(* CoDeSys 2.3.9.28 project: Aula08_ex2.pro *)
(* Libraries: Standard.lib 27.1.09 11:27:38, Util.lib 27.1.09 11:27:38, IecSfc.lib 24.11.08 08:07:15, SysLibTime.lib 27.1.09 11:27:38, SysTaskInfo.lib 24.11.08 08:07:15, SYSLIBCALLBACK.LIB 27.1.09 11:27:38 *)

(* PLC configuration (modules and I/O channels)
Hexswitch AT %IB0 [HexSwitch] rotary switch 0 = STOP, 1-15 = RUN
IOModules [CPX_MASTER] node 0, in %IB4 out %QB0
  8DI/8DO [CPX-8DI_8DO_Multi_I_O_module_1] node 0, in %IB4 out %QB0 {StringParam = 4,8,1,8,1; ByteParam = 7; ByteParam = 81; ByteParam = 0; ByteParam = 0; ByteParam = 0; ByteParam = 0; ByteParam = 0; IdleStateParam = 0; IdleModeParam = 255; IdleStateParam = 0; IdleModeParam = 255; IdleStateParam = 0; IdleModeParam = 255; IdleStateParam = 0; IdleModeParam = 255}
    AT %IB4 [ByteInput] -
    AT %QB0 [ByteOutput] -
  8DI/8DO [CPX-8DI_8DO_Multi_I_O_module_1] node 1, in %IB8 out %QB4 {StringParam = 4,8,1,8,1; ByteParam = 7; ByteParam = 81; ByteParam = 0; ByteParam = 0; ByteParam = 0; ByteParam = 0; ByteParam = 0; IdleStateParam = 0; IdleModeParam = 255; IdleStateParam = 0; IdleModeParam = 255; IdleStateParam = 0; IdleModeParam = 255; IdleStateParam = 0; IdleModeParam = 255}
    AT %IB8 [ByteInput] -
    AT %QB4 [ByteOutput] -
*)

(* Global variable list: Global_Variables *)
VAR_GLOBAL

	START AT %IX2.0 : BOOL;
	STOP AT %IX2.1 : BOOL;
	S1 AT %IX2.2 : BOOL;
	S2 AT %IX2.3 : BOOL;
	S3 AT %IX2.4 : BOOL;
	S4 AT %IX2.5 : BOOL;

	M1 AT %QX0.0 : BOOL;
	LP AT %QX0.1 : BOOL;
	C1 AT %QX0.2 : BOOL;
	C2 AT %QX0.3 : BOOL;

	MEM : BOOL;
	MEM2 : BOOL;
	MEM3: BOOL;
	MEM4: BOOL;
	MEM5: BOOL;

	T : TON;

END_VAR

(* POU PLC_PRG, LD *)
PROGRAM PLC_PRG
VAR

	T1: TON;
END_VAR
VAR (* helpers for the ST form of the networks *)
	_p1 : BOOL;
	_p2 : BOOL;
	_p3 : BOOL;
	_p4 : BOOL;
	_p5 : BOOL;
END_VAR
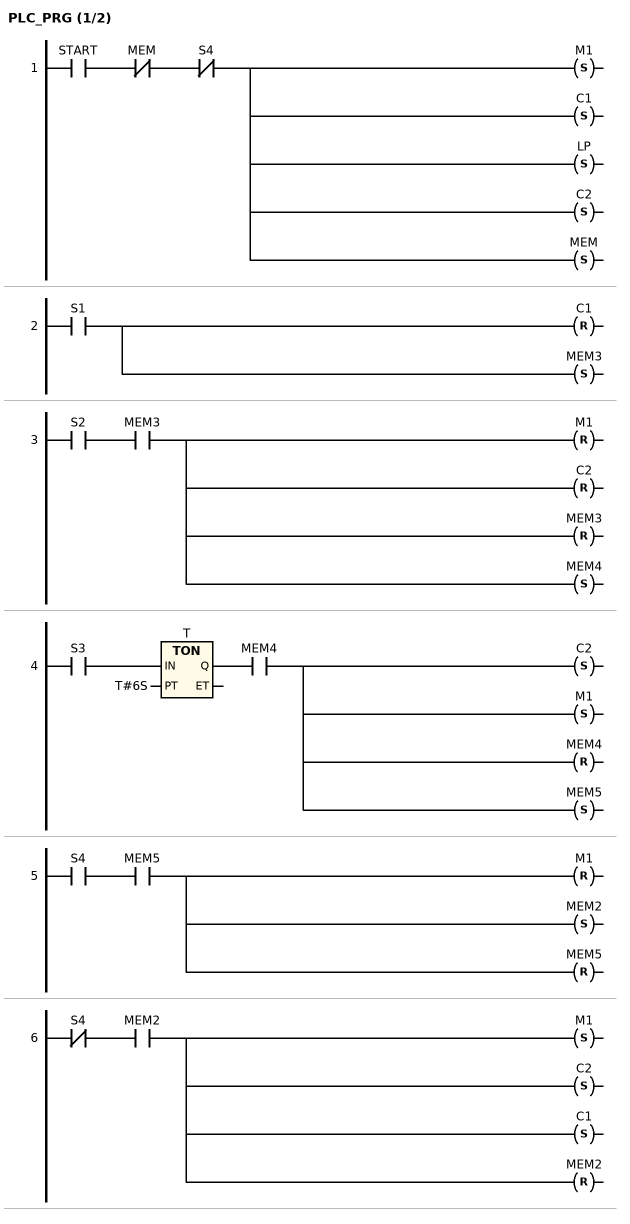
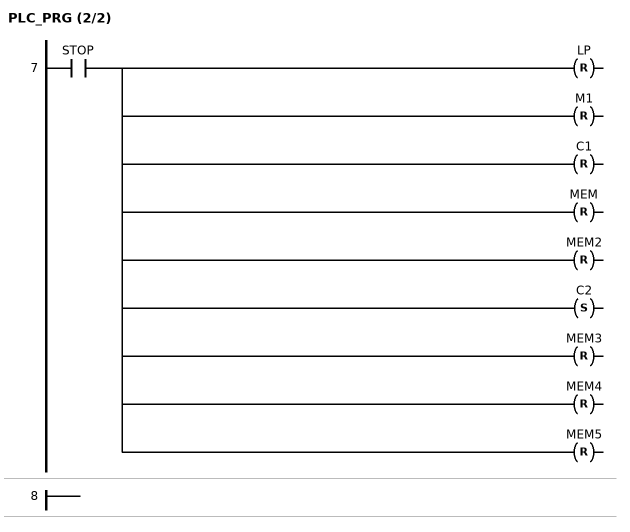
_LD_ (* Ladder Diagram *)
NETWORK 1
	[START] - [/MEM] - [/S4] --- (S M1) (S C1) (S LP) (S C2) (S MEM)
NETWORK 2
	[S1] --- (R C1) (S MEM3)
NETWORK 3
	[S2] - [MEM3] --- (R M1) (R C2) (R MEM3) (S MEM4)
NETWORK 4
	[S3] - T:TON(IN: *, PT: T#6S) - [MEM4] --- (S C2) (S M1) (R MEM4) (S MEM5)
NETWORK 5
	[S4] - [MEM5] --- (R M1) (S MEM2) (R MEM5)
NETWORK 6
	[/S4] - [MEM2] --- (S M1) (S C2) (S C1) (R MEM2)
NETWORK 7
	[STOP] --- (R LP) (R M1) (R C1) (R MEM) (R MEM2) (S C2) (R MEM3) (R MEM4) (R MEM5)
NETWORK 8
	*
_END_LD_
(* the same logic as Structured Text *)
(* Network 1 *)
_p1 := START AND NOT MEM AND NOT S4;
IF _p1 THEN M1 := TRUE; C1 := TRUE; LP := TRUE; C2 := TRUE; MEM := TRUE; END_IF;
(* Network 2 *)
IF S1 THEN C1 := FALSE; MEM3 := TRUE; END_IF;
(* Network 3 *)
_p2 := S2 AND MEM3;
IF _p2 THEN M1 := FALSE; C2 := FALSE; MEM3 := FALSE; MEM4 := TRUE; END_IF;
(* Network 4 *)
T(IN := S3, PT := T#6S);
_p3 := T.Q AND MEM4;
IF _p3 THEN C2 := TRUE; M1 := TRUE; MEM4 := FALSE; MEM5 := TRUE; END_IF;
(* Network 5 *)
_p4 := S4 AND MEM5;
IF _p4 THEN M1 := FALSE; MEM2 := TRUE; MEM5 := FALSE; END_IF;
(* Network 6 *)
_p5 := NOT S4 AND MEM2;
IF _p5 THEN M1 := TRUE; C2 := TRUE; C1 := TRUE; MEM2 := FALSE; END_IF;
(* Network 7 *)
IF STOP THEN LP := FALSE; M1 := FALSE; C1 := FALSE; MEM := FALSE; MEM2 := FALSE; C2 := TRUE; MEM3 := FALSE; MEM4 := FALSE; MEM5 := FALSE; END_IF;
(* Network 8 *)
END_PROGRAM
